// TIA Portal V18 export
TYPE "PartNumber_ShW"
// stored: IsFailsafeCompliant false
   STRUCT
      material_id : String[28];
      lot_code : String[18];
      Quantity : Int;
      ScanOK : Bool;
   END_STRUCT;
END_TYPE
